// TIA Portal V20 export
VAR_GLOBAL   // PLC tag table "LER_LVDT"
END_VAR
VAR_GLOBAL CONSTANT   // user constants
   ampNo : Int := 4;
END_VAR
